FUNCTION_BLOCK FB_AutoTrialRenew_ADS
VAR_INPUT
    bExpired            : BOOL;          // sygnał końca licencji (Twój)
    sProductId          : STRING(80);    // ID licencji Beckhoff
    sAdsServerNetId     : STRING(40);    // AMS ID serwera licencji
    nAdsServerPort      : UINT := 10000; // port ADS serwera
END_VAR

VAR_OUTPUT
    bBusy               : BOOL;
    bDone               : BOOL;
    bError              : BOOL;
    nErrorId            : UDINT;

    sLicenseOut         : STRING(1024);  // nowa licencja trial
END_VAR

VAR
    fbAdsWrite          : AdsWrite;
    fbAdsRead           : AdsRead;

    eState              : INT := 0;
    sBuffer             : STRING(1024);
END_VAR

// ============================================================================
//  STATE MACHINE
// ============================================================================
CASE eState OF

// ------------------------------------------------------
// IDLE
// ------------------------------------------------------
0:
    bBusy := FALSE;
    bDone := FALSE;
    bError := FALSE;

    IF bExpired THEN
        bBusy := TRUE;
        eState := 10;
    END_IF

// ------------------------------------------------------
// SEND REQUEST (ADS WRITE) – send ProductId to ADS server
// ------------------------------------------------------
10:
	fbAdsWrite(
		NETID	:=sAdsServerNetId,
		PORT	:=nAdsServerPort,
		IDXGRP	:=16#80000001,
		IDXOFFS	:=0,
		LEN		:=SIZEOF(sProductId),
		SRCADDR	:=ADR(sProductId),
		WRITE	:=TRUE);
		

    IF fbAdsWrite.ERR THEN
        bError := TRUE;
        nErrorId := fbAdsWrite.ERRID;
        eState := 0;

    ELSIF NOT fbAdsWrite.BUSY (*AND NOT fbAdsWrite.WRITE*) THEN
        eState := 20;
    END_IF

// ------------------------------------------------------
// GET TRIAL LICENCE (ADS READ)
// ------------------------------------------------------
20:
	fbAdsRead(
		NETID	:=sAdsServerNetId,
		PORT	:=nAdsServerPort, 
		IDXGRP	:=16#80000002,
		IDXOFFS	:=0,
		LEN		:=SIZEOF(sBuffer),
        DESTADDR:=ADR(sBuffer),
        READ	:=TRUE);
		
    IF fbAdsRead.ERR THEN
        bError := TRUE;
        nErrorId := fbAdsRead.ERRID;
        eState := 0;

    ELSIF NOT fbAdsRead.BUSY (*AND NOT fbAdsRead.READ *)THEN
        sLicenseOut := sBuffer;
        bDone := TRUE;
        bBusy := FALSE;
        eState := 0;
    END_IF

END_CASE

END_FUNCTION_BLOCK

(* stored: Version 1.2.0.0, ProductVersion 3.1.4026.13, FileIdentifier 07aaa83a60495c2e1b7c1b115645c497b132a7a6, FileSignature 59b7a5cfd298fe362f8743b3572c696e3077fb3e029877503aacdb567eadc7ac5330aece33efc528e5a4d6eb619e3b63105e1c7647337835341b1e712a724c277c3eee29082e1f3b3c4dd707709cb443e6a6e41371213165439bac1a2e4d73b8fa3b193cad16d9de4c65ad94a6a63f35298c1153dfd6a2fa379a908f44f5618e9bc0944861904daf08fa90c4fe94f8c1ca4721a9ff7fbbbf44b40928a9f69485279c4d408609ae41824174306592a4e216c954f615ea06e82f6cb5249ad3e1392ba8961d2c1eb40dd033977b0394480be8883f5162c12063d06be1530a5307974bbedf6a4fb4c4945138de84827f4a5ae3136ac47f862a4be170f6e64abfa382
   POU FB_AutoTrialRenew_ADS: Id {c79220c1-79e6-4401-9a40-b4c3162a208b}, SpecialFunc None *)
